(* IEC 61131-3 sources: K-ST/, 1 file *)

(* ---- try.st ---- *)
PROGRAM MAIN
VAR
   i : BOOL := TRUE;
END_VAR

IF i THEN
   EXIT;
END_IF;

END_PROGRAM
